// TIA Portal V17 export
// export: Created 2025-03-10T13:11:54.8361664Z, ExportSetting WithDefaults, DisplayName Totally Integrated Automation Portal, DisplayVersion V17 Update 8, DisplayName TIA Portal Openness, DisplayVersion V17 Update 8, DisplayName TIA Portal Version Control Interface, DisplayVersion V17, DisplayName SINAMICS Startdrive Advanced, DisplayVersion V17 SP2, DisplayName SINAMICS Startdrive G110M, G120, G120C, G120D, G120P, G115D, DisplayVersion V17 SP2, DisplayName SINAMICS Startdrive G130, G150, S120, S150, SINAMICS MV, S210, DisplayVersion V17 SP2, DisplayName STEP 7 Professional, DisplayVersion V17 Update 8, DisplayName SINUMERIK ONE STEP 7 Toolbox, DisplayVersion V17 Update 12, DisplayName SINUMERIK 840D sl STEP 7 Toolbox, DisplayVersion V17 Update 12, DisplayName STEP 7 Safety, DisplayVersion V17 Update 6, DisplayName WinCC Advanced, DisplayVersion V17 Update 8
TYPE "LBP_typeNCKProcessIRTFlags"
TITLE = LBP_NCKProcessIRT Output Interface / Interfaz de salida LBP_NCKProcessIRT / LBP_NCKProcessIRT Ausgangsschnittstelle
// User data type for LBP_NCKProcessIRT[FC3] Output Parameters / Tipo de datos de usuario para parámetros de salida LBP_NCKProcessIRT[FC3] / Anwender-Datentyp für LBP_NCKProcessIRT[FC3] Ausgangsparameter
// stored: IsFailsafeCompliant false
   STRUCT
      IRFromNck : Bool;   // Interrupt von NCK / Interrupt from NCK / Alarma de NCK
      TM : Bool;   // Werkzeugwechsel / Tool change / Cambio de herramienta
      InPosition : Array[1..31] of Bool;   // Achs- oder Spindelposition erreicht / Axis or spindle position reached / Posición de eje o cabezal alcanzada
      AuxFunction : Array[1..10] of Bool;   // Hilfsfunktion verfügbar / Auxiliary function available / Función auxiliar disponible
   END_STRUCT;
END_TYPE
